{attribute 'qualified_only'}
{attribute 'strict'}
TYPE E_Gamepad_Battery_Levels :
(
	// Battery is Empty or Unknown
	Empty := 0,
	// Battery is at low level
	Low := 1,
	// Battery is at medium level
	Medium := 2,
	// Battery is at full level
	Full := 3
);
END_TYPE

(* stored: Version 1.1.0.1, ProductVersion 3.1.4024.11
   DUT E_Gamepad_Battery_Levels: Id {8629e24e-2660-4f37-a73f-5543f84a5ff0} *)
